// TIA Portal V16 program export: 1 tag tables, 0 data types, 3 data blocks, 4 code blocks (in call order from the OBs), 4 instance data blocks

VAR_GLOBAL   // PLC tag table "Default tag table"
   tag1 AT %I0.0 : Bool;
   tag2 AT %I0.1 : Bool;
   tag3 AT %I0.2 : Bool;
END_VAR

DATA_BLOCK "Data"   // DB5
{ S7_Optimized_Access := 'TRUE' }
VERSION : 0.1
// stored: AutoNumber true, DBAccessibleFromOPCUA true, IsOnlyStoredInLoadMemory false, IsRetainMemResEnabled false, IsWriteProtectedInAS false, MemoryReserve 100
   VAR
      "Enable Serie" : Bool;
      Amplitud : Real;
      "Periodo (s)" : Real;
      N_Fourier : Int;
      "Serie f(t)" : Real;
   END_VAR
BEGIN
END_DATA_BLOCK

DATA_BLOCK "Data_Array"   // DB7
{ S7_Optimized_Access := 'TRUE' }
VERSION : 0.1
// stored: AutoNumber true, DBAccessibleFromOPCUA true, IsOnlyStoredInLoadMemory false, IsRetainMemResEnabled false, IsWriteProtectedInAS false, MemoryReserve 100
   VAR
      "E" : Array[0..1] of Real;
   END_VAR
BEGIN
END_DATA_BLOCK

DATA_BLOCK "Data_Sen"   // DB2
{ S7_Optimized_Access := 'TRUE' }
VERSION : 0.1
// stored: AutoNumber true, DBAccessibleFromOPCUA true, IsOnlyStoredInLoadMemory false, IsRetainMemResEnabled false, IsWriteProtectedInAS false, MemoryReserve 100
   VAR
      SenIN : Real;
      SenOUT : Real;
      SenCalc : Real;
   END_VAR
BEGIN
END_DATA_BLOCK

ORGANIZATION_BLOCK "Main"   // OB1, LAD, ProgramCycle
TITLE = "Main Program Sweep (Cycle)"
{ S7_Optimized_Access := 'TRUE' }
VERSION : 0.1
// stored: AutoNumber true, IsIECCheckEnabled false, SetENOAutomatically false
   VAR_INPUT
      Initial_Call : Bool;   // Initial call of this OB
      Remanence : Bool;   // =True, if remanent data are available
   END_VAR
BEGIN

REGION Network 1
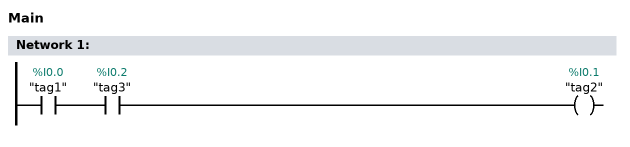
   RUNG wire#powerrail
      Contact( "tag1" )
      Contact( "tag3" )
      Coil( "tag2" )
   END_RUNG
   // the same network as SCL:
   "tag2" := "tag1" AND "tag3";
END_REGION
END_ORGANIZATION_BLOCK

ORGANIZATION_BLOCK "Cyclic interrupt"   // OB30, LAD, CyclicInterrupt
{ S7_Optimized_Access := 'TRUE' }
VERSION : 0.1
// stored: AutoNumber true, IsIECCheckEnabled false, SetENOAutomatically false
   VAR_INPUT
      Initial_Call : Bool;   // Initial call of this OB
      Event_Count : Int;   // Events discarded
   END_VAR
BEGIN

REGION Network 1
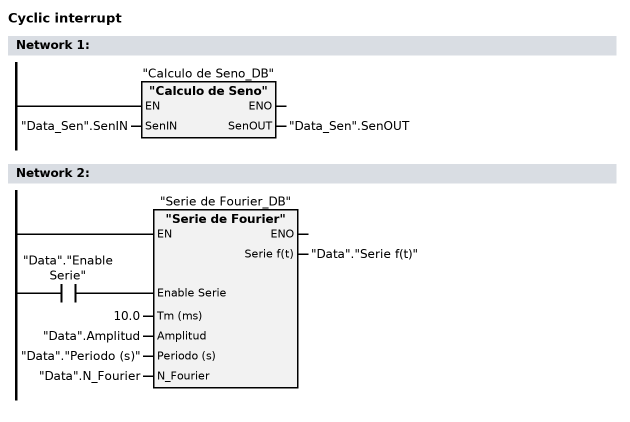
   RUNG wire#powerrail
      "Calculo de Seno_DB"(SenIN := "Data_Sen".SenIN, SenOUT => "Data_Sen".SenOUT)
   END_RUNG
   // the same network as SCL:
   "Calculo de Seno_DB"(SenIN := "Data_Sen".SenIN, SenOUT => "Data_Sen".SenOUT);   // "Calculo de Seno"
END_REGION

REGION Network 2
   RUNG wire#powerrail
      "Serie de Fourier_DB"("Enable Serie" := wire#w1, "Tm (ms)" := 10.0, Amplitud := "Data".Amplitud, "Periodo (s)" := "Data"."Periodo (s)", N_Fourier := "Data".N_Fourier, "Serie f(t)" => "Data"."Serie f(t)")
   END_RUNG
   RUNG wire#powerrail
      Contact( "Data"."Enable Serie" )
   END_RUNG wire#w1
   // the same network as SCL:
   "Serie de Fourier_DB"("Enable Serie" := "Data"."Enable Serie",   // "Serie de Fourier"
                         "Tm (ms)" := 10.0,
                         Amplitud := "Data".Amplitud,
                         "Periodo (s)" := "Data"."Periodo (s)",
                         N_Fourier := "Data".N_Fourier,
                         "Serie f(t)" => "Data"."Serie f(t)");
END_REGION
END_ORGANIZATION_BLOCK

FUNCTION_BLOCK "Calculo de Seno"   // FB1, LAD
{ S7_Optimized_Access := 'TRUE' }
VERSION : 0.1
// stored: AutoNumber true, IsIECCheckEnabled false, IsRetainMemResEnabled false, MemoryReserve 100, SetENOAutomatically false, UDAEnableTagReadback false
   VAR_OUTPUT
      SenOUT : Real;
   END_VAR
   VAR_IN_OUT
      SenIN : Real;
   END_VAR
   VAR
      Pulso1ms : Bool;
      AuxPulso1ms : Bool;
      AuxFlancoPulso4ms : Bool;
      Flanco4ms { ExternalAccessible := 'False'; ExternalVisible := 'False'; ExternalWritable := 'False'} : Bool;
   END_VAR
   VAR_TEMP
      SenAUX : Real;
      "SenIN-Radianes" : Real;
   END_VAR
   VAR CONSTANT
      PI : Real := 3.1416;
   END_VAR
BEGIN

REGION Network 1
   // Pasar de grados a radianes
END_REGION

REGION Network 2 (SCL)
   "Timer1".TON(IN := #AuxPulso1ms,
                PT := T#10ms,
                Q => #Pulso1ms);

   "Timer2".TOF(IN := NOT #Pulso1ms,
                PT := T#10ms,
                Q => #AuxPulso1ms);

   #Flanco4ms := NOT #Flanco4ms AND #Pulso1ms;

   IF #Pulso1ms THEN
       #SenIN := #SenIN + 1;
   END_IF;

   IF #SenIN >= 360.0 THEN
       #SenIN := 0.0;
   END_IF;

   #"SenIN-Radianes" := (#SenIN * #PI) / 180.0;

   #SenOUT := SIN(#"SenIN-Radianes");
END_REGION
END_FUNCTION_BLOCK

FUNCTION_BLOCK "Serie de Fourier"
{ S7_Optimized_Access := 'TRUE' }
VERSION : 0.1
   VAR_INPUT 
      "Enable Serie" : Bool;
      "Tm (ms)" : Real;
      Amplitud : Real;
      "Periodo (s)" : Real;
      N_Fourier : Int;
   END_VAR

   VAR_OUTPUT 
      "Serie f(t)" : Real;
   END_VAR

   VAR 
      cont { ExternalAccessible := 'False'; ExternalVisible := 'False'; ExternalWritable := 'False'} : Int;
   END_VAR

   VAR_TEMP 
      t : Real;
      n : Int;
      suma : Real;
   END_VAR

   VAR CONSTANT 
      PI : Real := 3.1416;
   END_VAR


BEGIN
	IF #"Enable Serie" THEN
	    //------------------------------Tiempo t(seg) en forma de puntos------------------------------
	    #cont := #cont + 1;
	    IF #cont > REAL_TO_INT(1000 * #"Periodo (s)" / #"Tm (ms)") THEN // Si cont > Periodo en forma de puntos
	        #cont := 0;
	    END_IF;
	    
	    #t := #cont * #"Tm (ms)" / 1000.0; //tiempo t en (seg)
	    
	    //------------Serie de Fourier------------
	    FOR #n := 1 TO #N_Fourier DO
	        IF #"Enable Serie" = TRUE THEN
	            //Onda Completa
	            #suma := #suma + (COS(#n * 2 * #PI * #t / #"Periodo (s)")) / (4 * SQRT(#n) - 1); //Sumatoria infinita
	        ELSE
	            #suma := 0;
	        END_IF;
	        
	    END_FOR;
	    
	    IF #"Enable Serie" = TRUE THEN
	        //Onda Completa
	        #"Serie f(t)" := (2 * #Amplitud / #PI) - (4 * #Amplitud / #PI) * #suma; //
	    ELSE
	        #"Serie f(t)" := 0;
	    END_IF;
	ELSE
	    
	    #t := 0;
	    #suma:=0;
	    #"Serie f(t)" := 0;
	  
	END_IF;
	
	
	    
	
	
	    
	
	
	
END_FUNCTION_BLOCK

DATA_BLOCK "Calculo de Seno_DB"   // DB1
VERSION : 0.1
// stored: AutoNumber true, DBAccessibleFromOPCUA true, InstanceOfName Calculo de Seno, InstanceOfType FB
"Calculo de Seno"
BEGIN
END_DATA_BLOCK

DATA_BLOCK "Serie de Fourier_DB"   // DB6
VERSION : 0.1
// stored: AutoNumber true, DBAccessibleFromOPCUA true, InstanceOfName Serie de Fourier, InstanceOfType FB
"Serie de Fourier"
BEGIN
END_DATA_BLOCK

DATA_BLOCK "Timer1"   // DB3
{ S7_Optimized_Access := 'TRUE' }
// stored: AutoNumber true, DBAccessibleFromOPCUA true, InstanceOfName IEC_TIMER, OfSystemLibElement IEC_TIMER, OfSystemLibVersion 1.0
"IEC_TIMER"
   // VAR
   //    PT : Time;
   //    ET { ExternalWritable := 'False'} : Time;
   //    IN : Bool;
   //    Q { ExternalWritable := 'False'} : Bool;
   // END_VAR
BEGIN
END_DATA_BLOCK

DATA_BLOCK "Timer2"   // DB4
{ S7_Optimized_Access := 'TRUE' }
// stored: AutoNumber true, DBAccessibleFromOPCUA true, InstanceOfName IEC_TIMER, OfSystemLibElement IEC_TIMER, OfSystemLibVersion 1.0
"IEC_TIMER"
   // VAR
   //    PT : Time;
   //    ET { ExternalWritable := 'False'} : Time;
   //    IN : Bool;
   //    Q { ExternalWritable := 'False'} : Bool;
   // END_VAR
BEGIN
END_DATA_BLOCK
